SUBAPPLICATION Uebung_070_AX (* WBSD auf UT ausgeben *)
  (* Standard: 61499-2; Description: Copyright (c) 2023 Meisterschulen am Ostbahnhof This program and the accompanying materials are made available under the terms of the Eclipse Public License 2.0 which is available at https://www.eclipse.org/legal/epl-2.0/ SPDX-License-Identifier: EPL-2.0 *)
  (* Version 1.0, 2023-10-23, Franz Höpfinger, Meisterschulen am Ostbahnhof, initial API and implementation and/or initial documentation *)
  PACKAGE Uebungen;
  IMPORT Uebungen::const::UT::TECU::DefaultPool_TECU::NumberVariable_Wheel_based_machine_speed;
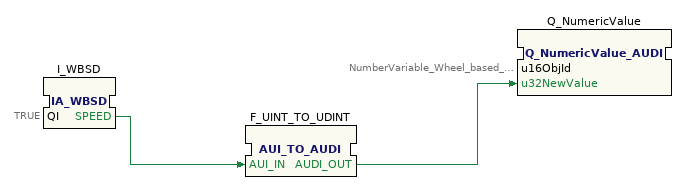
  FBS
    I_WBSD : isobus::tecu::IA_WBSD(QI := TRUE);
    Q_NumericValue : isobus::UT::Q::Q_NumericValue_AUDI(u16ObjId := NumberVariable_Wheel_based_machine_speed);
    F_UINT_TO_UDINT : adapter::conversion::unidirectional::AUI_TO_AUDI;
  END_FBS
  ADAPTER_CONNECTIONS
    I_WBSD.SPEED TO F_UINT_TO_UDINT.AUI_IN;
    F_UINT_TO_UDINT.AUDI_OUT TO Q_NumericValue.u32NewValue;
  END_CONNECTIONS
END_SUBAPPLICATION
